TYPE TYP_HW_L4000 :
STRUCT
	In : TYP_HW_L4000_IN;
	Out : TYP_HW_L4000_OUT;
END_STRUCT
END_TYPE

(* stored: Version 1.1.0.1, ProductVersion 3.1.4024.12
   DUT TYP_HW_L4000: Id {effc9be8-3e0c-4878-afe8-fb53a2926daa} *)
